TYPE CmpSafetyInterfaceConv :
STRUCT

	//Station to Main Safety interface
	// Currently no data flows back from stn to Main saftey interface
	
	//Main Safety interface to Station
	iSafetyResetPB: BOOL;		 
	iSafetyCtrlGroupError: BOOL;	
	iEstopRlyTripped: BOOL;				
	iEstopButtonNOK1: BOOL;		
	iAirPressureOk: BOOL;
	
END_STRUCT

END_TYPE

(* stored: Version 1.1.0.1, ProductVersion 3.1.4024.6
   DUT CmpSafetyInterfaceConv: Id {02099a9a-919c-4d0e-9052-70b07fa7389f} *)
